// Mitsubishi GX Works2 project: code mau hmi_plc2n 20mr   PLC: FX2N/FX2NC

PROGRAM MAIN
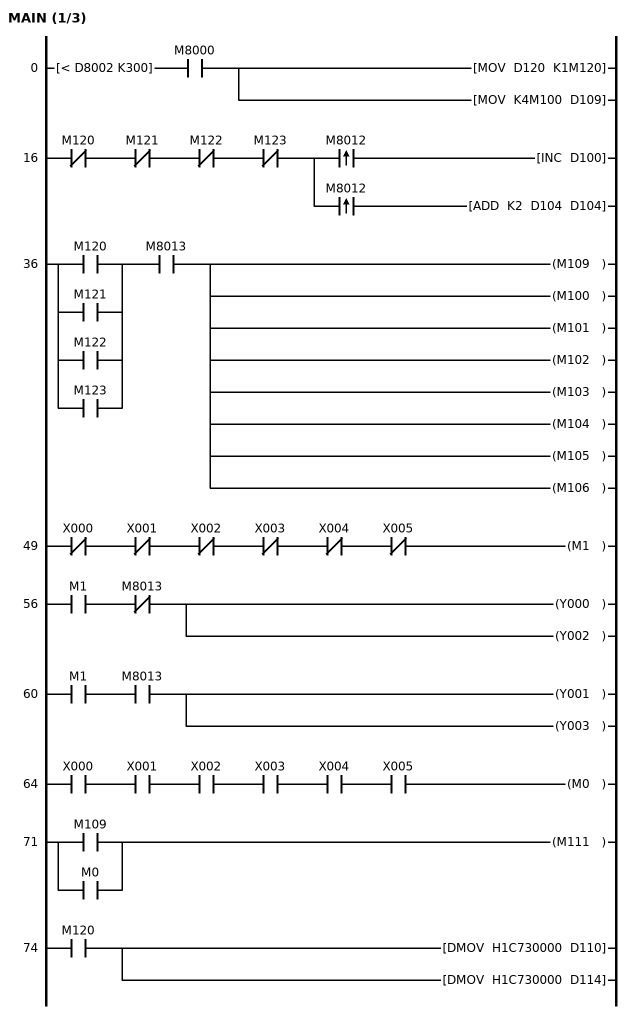
0     LD<     D8002 K300
      AND     M8000
      MOV     D120 K1M120
      MOV     K4M100 D109
16    LDI     M120
      ANI     M121
      ANI     M122
      ANI     M123
      MPS
      ANDP    M8012
      INC     D100
      MPP
      ANDP    M8012
      ADD     K2 D104 D104
36    LD      M120
      OR      M121
      OR      M122
      OR      M123
      AND     M8013
      OUT     M109
      OUT     M100
      OUT     M101
      OUT     M102
      OUT     M103
      OUT     M104
      OUT     M105
      OUT     M106
49    LDI     X000
      ANI     X001
      ANI     X002
      ANI     X003
      ANI     X004
      ANI     X005
      OUT     M1
56    LD      M1
      ANI     M8013
      OUT     Y000
      OUT     Y002
60    LD      M1
      AND     M8013
      OUT     Y001
      OUT     Y003
64    LD      X000
      AND     X001
      AND     X002
      AND     X003
      AND     X004
      AND     X005
      OUT     M0
71    LD      M109
      OR      M0
      OUT     M111
74    LD      M120
      DMOV    H1C730000 D110
      DMOV    H1C730000 D114
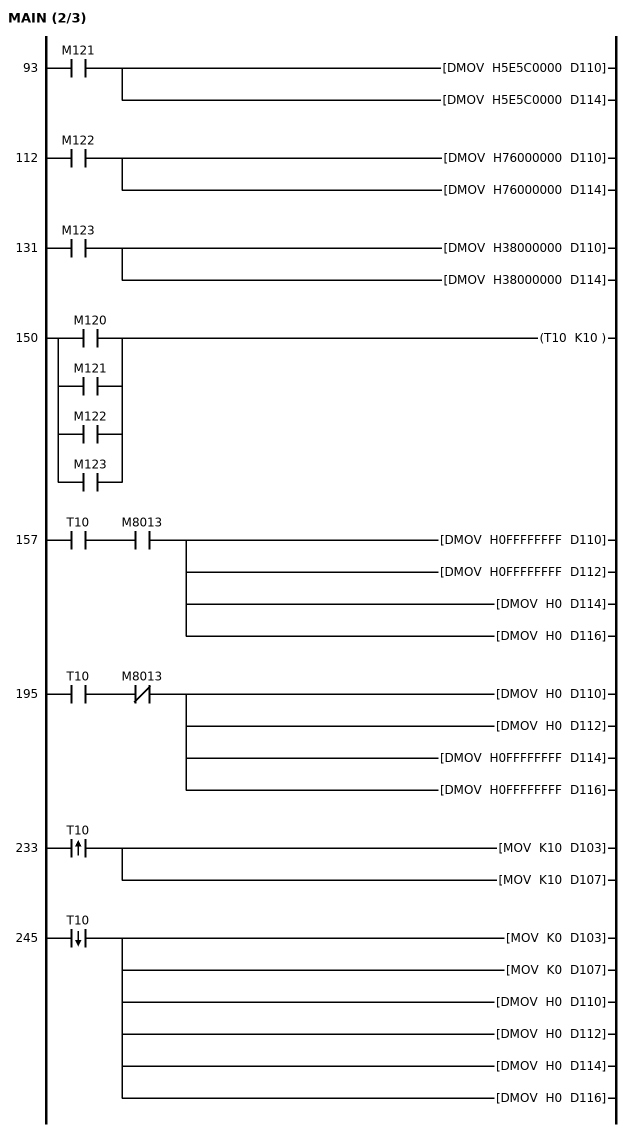
93    LD      M121
      DMOV    H5E5C0000 D110
      DMOV    H5E5C0000 D114
112   LD      M122
      DMOV    H76000000 D110
      DMOV    H76000000 D114
131   LD      M123
      DMOV    H38000000 D110
      DMOV    H38000000 D114
150   LD      M120
      OR      M121
      OR      M122
      OR      M123
      OUT     T10 K10
157   LD      T10
      AND     M8013
      DMOV    H0FFFFFFFF D110
      DMOV    H0FFFFFFFF D112
      DMOV    H0 D114
      DMOV    H0 D116
195   LD      T10
      ANI     M8013
      DMOV    H0 D110
      DMOV    H0 D112
      DMOV    H0FFFFFFFF D114
      DMOV    H0FFFFFFFF D116
233   LDP     T10
      MOV     K10 D103
      MOV     K10 D107
245   LDF     T10
      MOV     K0 D103
      MOV     K0 D107
      DMOV    H0 D110
      DMOV    H0 D112
      DMOV    H0 D114
      DMOV    H0 D116
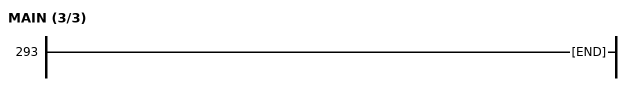
293   END
END_PROGRAM
